# EPICS autosave request: ADApp/Db/NDFileHDF5_settings.req
$(P)$(R)NumRowChunks
$(P)$(R)NumColChunks
$(P)$(R)NumFramesChunks
$(P)$(R)BoundaryAlign
$(P)$(R)BoundaryThreshold
$(P)$(R)NumFramesFlush
$(P)$(R)Compression
$(P)$(R)NumDataBits
$(P)$(R)DataBitsOffset
$(P)$(R)SZipNumPixels
$(P)$(R)ZLevel
$(P)$(R)StorePerform
$(P)$(R)StoreAttr
$(P)$(R)StrAttrDataType
$(P)$(R)NumExtraDims
$(P)$(R)ExtraDimSizeN
$(P)$(R)ExtraDimSizeX
$(P)$(R)ExtraDimSizeY
$(P)$(R)XMLFileName
file "NDPluginFile_settings.req", P=$(P), R=$(R)
